{attribute 'qualified_only'}
VAR_GLOBAL
	//Grille d'où sont passé les robots adverses
	grid : ARRAY [0..5] OF ARRAY [0..8] OF BOOL;
	//Reset de la grille dans le raspberry pi
	reset : BOOL;
END_VAR

(* stored: Version 1.1.0.1, ProductVersion 3.1.4024.12
   GVL G_RPI: Id {f35cac2b-5fa6-4657-a29d-7bdda37b36c6} *)
